FUNCTION_BLOCK T_Axis EXTENDS T_NamedBase IMPLEMENTS I_Axis
VAR
END_VAR

END_FUNCTION_BLOCK

(* stored: Version 1.1.0.1, ProductVersion 3.1.4024.12
   POU T_Axis: Id {738671f0-e5f5-41d5-a646-52cb8f1590cf}, SpecialFunc None *)
